(* PLC project SafeLOGIC-1, BrAutomation SafeDESIGNER  4.3.4.4 *)
(* stored: companyURL http://www.br-automation.com, creationDateTime Thu Jun 24 15:36:39 2021 *)

PROGRAM Main
  VAR  (* added by the conversion: wires and edge detectors of the diagram *)
    _SAFEBOOL_TO_BOOL20_OUT : BOOL;
  END_VAR

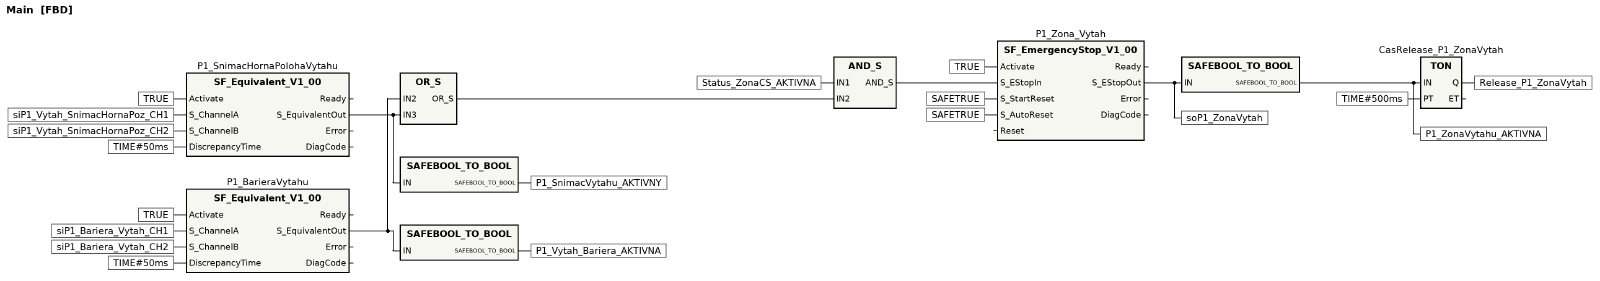
(* FBD diagram, written out as Structured Text *)
P1_BarieraVytahu(Activate := TRUE, S_ChannelA := siP1_Bariera_Vytah_CH1, S_ChannelB := siP1_Bariera_Vytah_CH2, DiscrepancyTime := TIME#50ms);
P1_SnimacHornaPolohaVytahu(Activate := TRUE, S_ChannelA := siP1_Vytah_SnimacHornaPoz_CH1, S_ChannelB := siP1_Vytah_SnimacHornaPoz_CH2, DiscrepancyTime := TIME#50ms);
P1_Zona_Vytah(Activate := TRUE, S_EStopIn := AND_S(Status_ZonaCS_AKTIVNA, OR_S(P1_BarieraVytahu.S_EquivalentOut, P1_SnimacHornaPolohaVytahu.S_EquivalentOut)), S_StartReset := SAFETRUE, S_AutoReset := SAFETRUE);
soP1_ZonaVytah := P1_Zona_Vytah.S_EStopOut;
_SAFEBOOL_TO_BOOL20_OUT := SAFEBOOL_TO_BOOL(P1_Zona_Vytah.S_EStopOut);
P1_ZonaVytahu_AKTIVNA := _SAFEBOOL_TO_BOOL20_OUT;
CasRelease_P1_ZonaVytah(IN := _SAFEBOOL_TO_BOOL20_OUT, PT := TIME#500ms);
Release_P1_ZonaVytah := CasRelease_P1_ZonaVytah.Q;
P1_Vytah_Bariera_AKTIVNA := SAFEBOOL_TO_BOOL(P1_BarieraVytahu.S_EquivalentOut);
P1_SnimacVytahu_AKTIVNY := SAFEBOOL_TO_BOOL(P1_SnimacHornaPolohaVytahu.S_EquivalentOut);
END_PROGRAM
